             ELSIF (#instMoveSuperimposed.Error = TRUE) THEN
               // Errorhandling
               #statStatus := #ERR_MC_MOVESUPERIMPOSED;
               #statStatusText := STRING#'ERR_MC_MOVESUPERIMPOSED';
               #statErrorAutoCleared := TRUE;
               #statDiagnostics.subfunctionStatus := #statSubfunctionStatus := #instMoveSuperimposed.ErrorID;
               // Set next state
               #statFBState := #AXIS_STOP_ON_ERROR_SELECTION;
               #statSupImpMotionState := #NO_SELECTION;
             ELSE
               ; // command selected
             END_IF;
             #statExeOfSupImpMotionState := 16#0;
             #statExeOfSupImpMotionState.%X0 := #instMoveSuperimposed.Busy;
             #statExeOfSupImpMotionState.%X1 := #instMoveSuperimposed.Done;
             #statExeOfSupImpMotionState.%X2 := #instMoveSuperimposed.CommandAborted;
             #statExeOfSupImpMotionState.%X3 := #instMoveSuperimposed.Error;
             #statExeOfSupImpMotionState.%X4 := #instMoveSuperimposed.Busy;
           END_IF;
         END_REGION

       #PHASING_SELECTED:
         // Additional features (applicative) : Change setpoint on the fly (phaseShift)
         REGION PHASING_SELECTED
           // Firstcycle of command
           IF (#statFirstCycleSupImpMotion = TRUE) THEN
             // Reset MC_PHASING_ABSOLUTE command
             #instPhasingAbsolute(Master := #master,
                                  Slave := #statAxis,
                                  Execute := FALSE);

             // Reset MC_PHASING_RELATIVE command
             #instPhasingRelative(Master := #master,
                                  Slave := #statAxis,
                                  Execute := FALSE);

             #statPhaseShift := #configuration.phasing.phaseShift;
             #statSupImpVelocity := #configuration.phasing.velocity;
             #statSupImpAcceleration := #configuration.phasing.acceleration;
             #statSupImpDeceleration := #configuration.phasing.deceleration;
             #statSupImpJerk := #configuration.phasing.jerk;
             #statSupImpProfileReference := #configuration.phasing.profileReference;
             #statSupImpDistance := #configuration.phasing.phasingDistance;
             #statSupImpStartPosition := #configuration.phasing.startPosition;
             #statSupImpDirection := #configuration.phasing.direction;

             #statPhaseAbsolute := #configuration.phasing.phaseAbsolute;
             #statChangePhaseShiftOnTheFly := #configuration.phasing.phaseShiftChangeOnTheFly;

           ELSIF ((#statChangePhaseShiftOnTheFly = TRUE) AND
             (#configuration.phasing.phaseShift <> #statPhaseShift))
             AND (#statPhaseAbsolute = TRUE)
             AND (#instPhasingAbsolute.CommandAborted = FALSE)
           THEN
             // Reset MC_PHASING_ABSOLUTE command - Phaseshift on the fly is only possible at phasing absolut
             #instPhasingAbsolute(Master := #master,
                                  Slave := #statAxis,
                                  Execute := FALSE);

             #statPhaseShift := #configuration.phasing.phaseShift;

             // V1.0.5 Copy also Dynamics
             #statSupImpVelocity := #configuration.phasing.velocity;
             #statSupImpAcceleration := #configuration.phasing.acceleration;
             #statSupImpDeceleration := #configuration.phasing.deceleration;
             #statSupImpJerk := #configuration.phasing.jerk;
             #statSupImpProfileReference := #configuration.phasing.profileReference;
             #statSupImpDistance := #configuration.phasing.phasingDistance;
             #statSupImpStartPosition := #configuration.phasing.startPosition;
             #statSupImpDirection := #configuration.phasing.direction;

           END_IF;

           // Select phasing absolut or relative 
           IF (#statPhaseAbsolute = TRUE) THEN
             // Absolute phasing
             // Call MC_Command
             #instPhasingAbsolute(Master := #master,
                                  Slave := #statAxis,
                                  Execute := #statSupImpCommand.%X1, // Input: phasing
                                  PhaseShift := #statPhaseShift,
                                  Velocity := #statSupImpVelocity,
                                  Acceleration := #statSupImpAcceleration,
                                  Deceleration := #statSupImpDeceleration,
                                  Jerk := #statSupImpJerk,
                                  ProfileReference := #statSupImpProfileReference,
                                  PhasingDistance := #statSupImpDistance,
                                  StartPosition := #statSupImpStartPosition,
                                  Direction := #statSupImpDirection);

             // Evaluate MC_Command
             IF (#instPhasingAbsolute.Busy = FALSE) AND
               (#instPhasingAbsolute.Error = FALSE) AND
               (#instPhasingAbsolute.Done = FALSE) AND
               (#instPhasingAbsolute.CommandAborted = FALSE)
             THEN
               // Return to NO_SELECTION if command finished
               #statSupImpMotionState := #NO_SELECTION;

             ELSIF (#instPhasingAbsolute.Error = TRUE) THEN
               // Errorhandling
               #statStatus := #ERR_MC_PHASINGABSOLUTE;
               #statStatusText := STRING#'ERR_MC_PHASINGABSOLUTE';
               #statErrorAutoCleared := TRUE;
               #statDiagnostics.subfunctionStatus := #statSubfunctionStatus := #instPhasingAbsolute.ErrorID;
               #statChangePhaseShiftOnTheFly := FALSE;
               // Set next state
               #statFBState := #AXIS_STOP_ON_ERROR_SELECTION;
               #statSupImpMotionState := #NO_SELECTION;
             ELSE
               ; // Command busy
             END_IF;
             #statExeOfSupImpMotionState := 16#0;
             #statExeOfSupImpMotionState.%X0 := #instPhasingAbsolute.Busy;
             #statExeOfSupImpMotionState.%X1 := #instPhasingAbsolute.Done;
             #statExeOfSupImpMotionState.%X2 := #instPhasingAbsolute.CommandAborted;
             #statExeOfSupImpMotionState.%X3 := #instPhasingAbsolute.Error;
             #statExeOfSupImpMotionState.%X4 := #instPhasingAbsolute.StartPhasing;
           ELSE
             // Relative phasing  
             // Call MC_Command
             #instPhasingRelative(Master := #master,
                                  Slave := #statAxis,
                                  Execute := #statSupImpCommand.%X1, // Input: phasing
                                  PhaseShift := #statPhaseShift,
                                  Velocity := #statSupImpVelocity,
                                  Acceleration := #statSupImpAcceleration,
                                  Deceleration := #statSupImpDeceleration,
                                  Jerk := #statSupImpJerk,
                                  ProfileReference := #configuration.phasing.profileReference,
                                  PhasingDistance := #configuration.phasing.phasingDistance,
                                  StartPosition := #configuration.phasing.startPosition,
                                  Direction := #configuration.phasing.direction);

             // Evaluate MC_Command
             IF (#instPhasingRelative.Busy = FALSE) AND
               (#instPhasingRelative.Error = FALSE) AND
               (#instPhasingRelative.Done = FALSE) AND
               (#instPhasingRelative.CommandAborted = FALSE)
             THEN
               // Return to NO_SELECTION if command finished
               #statSupImpMotionState := #NO_SELECTION;

             ELSIF (#instPhasingRelative.Error = TRUE) THEN
               // Errorhandling
               #statStatus := #ERR_MC_PHASINGRELATIVE;
               #statStatusText := STRING#'ERR_MC_PHASINGRELATIVE';
               #statErrorAutoCleared := TRUE;
               #statDiagnostics.subfunctionStatus := #statSubfunctionStatus := #instPhasingRelative.ErrorID;
               #statChangePhaseShiftOnTheFly := FALSE;
               // Set next state
               #statFBState := #AXIS_STOP_ON_ERROR_SELECTION;
               #statSupImpMotionState := #NO_SELECTION;
             ELSE
               ; // Command selected
             END_IF;
             #statExeOfSupImpMotionState := 16#0;
             #statExeOfSupImpMotionState.%X0 := #instPhasingRelative.Busy;
             #statExeOfSupImpMotionState.%X1 := #instPhasingRelative.Done;
             #statExeOfSupImpMotionState.%X2 := #instPhasingRelative.CommandAborted;
             #statExeOfSupImpMotionState.%X3 := #instPhasingRelative.Error;
             #statExeOfSupImpMotionState.%X4 := #instPhasingRelative.StartPhasing;
           END_IF;
         END_REGION

       #OFFSET_SELECTED:
         REGION OFFSET_SELECTED
           // Firstcycle of command
           IF (#statFirstCycleSupImpMotion = TRUE) THEN
             // Reset MC_OFFSET_ABSOLUTE command
             #instOffsetAbsolute(Slave := #statAxis,
                                 Execute := FALSE);

             // Reset MC_OFFSET_RELATIVE command
             #instOffsetRelative(Slave := #statAxis,
                                 Execute := FALSE);

             #statOffsetValue := #configuration.offset.offset;
             #statSupImpProfileReference := #configuration.offset.profileReference;
             #statSupImpDistance := #configuration.offset.offsetDistance;
             #statSupImpStartPosition := #configuration.offset.startPosition;
             #statSupImpDirection := #configuration.offset.direction;

             #statOffsetAbsolute := #configuration.offset.offsetAbsolute;
             #statChangeOffsetOnTheFly := #configuration.offset.offsetChangeOnTheFly;

           ELSIF ((#statChangeOffsetOnTheFly = TRUE) AND
             (#configuration.offset.offset <> #statOffsetValue))
             AND (#statOffsetAbsolute = TRUE)
             AND (#instOffsetAbsolute.CommandAborted = FALSE)
           THEN
             // Reset MC_OFFSET_ABSOLUTE command - Offset on the fly is only possible at phasing absolut
             #instOffsetAbsolute(Slave := #statAxis,
                                 Execute := FALSE);

             #statOffsetValue := #configuration.offset.offset;
           END_IF;

           // Select offset absolut or relative 
           IF (#statOffsetAbsolute = TRUE) THEN
             // Absolute phasing
             // Call MC_Command
             #instOffsetAbsolute(Slave := #statAxis,
                                 Execute := #statSupImpCommand.%X2, // Input: offset
                                 Offset := #statOffsetValue,
                                 ProfileReference := #statSupImpProfileReference,
                                 OffsetDistance := #statSupImpDistance,
                                 StartPosition := #statSupImpStartPosition,
                                 Direction := #statSupImpDirection);

             // Evaluate MC_Command
             IF (#instOffsetAbsolute.Busy = FALSE) AND
               (#instOffsetAbsolute.Error = FALSE) AND
               (#instOffsetAbsolute.Done = FALSE) AND
               (#instOffsetAbsolute.CommandAborted = FALSE)
             THEN
               // Return to NO_SELECTION if command finished
               #statSupImpMotionState := #NO_SELECTION;

             ELSIF (#instOffsetAbsolute.Error = TRUE) THEN
               // Errorhandling
               #statStatus := #ERR_MC_OFFSETABSOLUTE;
               #statStatusText := STRING#'ERR_MC_OFFSETABSOLUTE';
               #statErrorAutoCleared := TRUE;
               #statDiagnostics.subfunctionStatus := #statSubfunctionStatus := #instOffsetAbsolute.ErrorID;
               #statChangeOffsetOnTheFly := FALSE;
               // Set next state
               #statFBState := #AXIS_STOP_ON_ERROR_SELECTION;
               #statSupImpMotionState := #NO_SELECTION;
             ELSE
               ; // Command busy
             END_IF;
             #statExeOfSupImpMotionState := 16#0;
             #statExeOfSupImpMotionState.%X0 := #instOffsetAbsolute.Busy;
             #statExeOfSupImpMotionState.%X1 := #instOffsetAbsolute.Done;
             #statExeOfSupImpMotionState.%X2 := #instOffsetAbsolute.CommandAborted;
             #statExeOfSupImpMotionState.%X3 := #instOffsetAbsolute.Error;
             #statExeOfSupImpMotionState.%X4 := #instOffsetAbsolute.StartOffset;
           ELSE
             // Relative offset  
             // Call MC_Command
             #instOffsetRelative(Slave := #statAxis,
                                 Execute := #statSupImpCommand.%X2, // Input: offset
                                 Offset := #statOffsetValue,
                                 ProfileReference := #configuration.offset.profileReference,
                                 OffsetDistance := #configuration.offset.offsetDistance,
                                 StartPosition := #configuration.offset.startPosition,
                                 Direction := #configuration.offset.direction);

             // Evaluate MC_Command
             IF (#instOffsetRelative.Busy = FALSE) AND
               (#instOffsetRelative.Error = FALSE) AND
               (#instOffsetRelative.Done = FALSE) AND
               (#instOffsetRelative.CommandAborted = FALSE)
             THEN
               // Return to NO_SELECTION if command finished
               #statSupImpMotionState := #NO_SELECTION;

             ELSIF (#instOffsetRelative.Error = TRUE) THEN
               // Errorhandling
               #statStatus := #ERR_MC_OFFSETRELATIVE;
               #statStatusText := STRING#'ERR_MC_OFFSETRELATIVE';
               #statErrorAutoCleared := TRUE;
               #statDiagnostics.subfunctionStatus := #statSubfunctionStatus := #instOffsetRelative.ErrorID;
               #statChangeOffsetOnTheFly := FALSE;
               // Set next state
               #statFBState := #AXIS_STOP_ON_ERROR_SELECTION;
               #statSupImpMotionState := #NO_SELECTION;
             ELSE
               ; // Command selected
             END_IF;
             #statExeOfSupImpMotionState := 16#0;
             #statExeOfSupImpMotionState.%X0 := #instOffsetRelative.Busy;
             #statExeOfSupImpMotionState.%X1 := #instOffsetRelative.Done;
             #statExeOfSupImpMotionState.%X2 := #instOffsetRelative.CommandAborted;
             #statExeOfSupImpMotionState.%X3 := #instOffsetRelative.Error;
             #statExeOfSupImpMotionState.%X4 := #instOffsetRelative.StartOffset;
           END_IF;
         END_REGION
       ELSE
         // Errorhandling
         #statStatus := #ERR_UNDEFINED_SUPERIMPOSED_MOTION_STATE;
         #statStatusText := STRING#'ERR_UNDEFINED_SUPERIMPOSED_MOTION_STATE';
         #statErrorUserCleared := TRUE;
         #statDiagnostics.subfunctionStatus := #statSubfunctionStatus := 0;
         // Set errorstate
         #statFBState := #FB_ERROR;
     END_CASE;
   END_REGION

   //----------------------------------------------------------------------------------------------
   // Execution of torquelimiting functionality
   //----------------------------------------------------------------------------------------------
   REGION EXECUTION_OF_TORQUELIMTING
     // Statemachine for torquelimiting 
     REPEAT
       #tempStateChangeActive := FALSE;
       CASE #statTorqueLimitingState OF
         #NO_TORQUE_LIMITING_ACTIVE:
           ;

         #TORQUE_LIMITING_DISABLE:
           // Torquelimiting disable
           #instTorqueLimiting(Axis := #statAxis,
                               Enable := FALSE);

           // Check state of torque limting
           IF (#instTorqueLimiting.Busy = FALSE)
           THEN
             // set next state
             #statTorqueLimitingState := #NO_TORQUE_LIMITING_ACTIVE;
           ELSE
             ; // Waiting for MC_Torquelimiting is not busy
           END_IF;

         #TORQUE_LIMTING_SELECTED:
           // No extended homing function active
           #instTorqueLimiting(Axis := #statAxis,
                               Enable := #statExtendedCommand.%X1,
                               Limit := #configuration.torqueLimiting.limit,
                               Mode := #configuration.torqueLimiting.mode);

           IF (#instTorqueLimiting.Busy = FALSE) THEN
             // Reset state
             #statTorqueLimitingState := #NO_TORQUE_LIMITING_ACTIVE;
           END_IF;

         #FIXED_STOP_DETECTION_ACTIVE:
           // Extended homing function active
           #instTorqueLimiting(Axis := #statAxis,
                               Enable := TRUE,
                               Limit := #configuration.homing.extendedModeTorqueLimit, // V01.00.03 Always use configured value
                               Mode := #MODE_FIXED_STOP_DETECTION);

           IF ((#statHomingSubState = #HOMING_IDLE) AND (#statBasicMotionState = #ACTIVE_HOMING_SELECTED))
           THEN
             // Fixed stop process has finished - Axis is still in clamping
             #statTorqueLimitingState := #FIXED_STOP_DETECTION_FINISHED;
             #tempStateChangeActive := TRUE;

           ELSIF (#statBasicMotionState <> #ACTIVE_HOMING_SELECTED)
           THEN
             // Error occurred - change state depending on inClamping
             IF (#instTorqueLimiting.InClamping = TRUE)
             THEN
               // Axis is in clamping
               #statTorqueLimitingState := #FIXED_STOP_DETECTION_ERROR_IN_CLAMPING;
               #tempStateChangeActive := TRUE;
             ELSE
               // Axis is in not clamping
               #statTorqueLimitingState := #FIXED_STOP_DETECTION_ERROR_NOT_IN_CLAMPING;
               #tempStateChangeActive := TRUE;
             END_IF;
           ELSE
             ; // Fixed stop detection is running
           END_IF;

         #FIXED_STOP_DETECTION_FINISHED:
           // Homing on fixed stop process has finished
           #instTorqueLimiting(Axis := #statAxis,
                               Enable := TRUE,
                               Limit := #configuration.homing.extendedModeTorqueLimit, // V01.00.03 Always use configured value
                               Mode := #MODE_FIXED_STOP_DETECTION);

           IF (#instTorqueLimiting.InClamping = FALSE)
           THEN
             // InClamping = FALSE
             IF (#statExtendedCommand.%X1 = TRUE) // Torquelimiting
             THEN
               #statTorqueLimitingState := #TORQUE_LIMTING_SELECTED;
             ELSE
               #statTorqueLimitingState := #TORQUE_LIMITING_DISABLE;
             END_IF;
             #tempStateChangeActive := TRUE;
           ELSE
             // InClamping = TRUE
             IF (#statExtendedCommand.%X1 = TRUE) // Torquelimiting
               AND (#configuration.torqueLimiting.mode = #MODE_FIXED_STOP_DETECTION)
             THEN
               // Change State
               #statTorqueLimitingState := #TORQUE_LIMTING_SELECTED;
               #tempStateChangeActive := TRUE;
             ELSE
               ; // Wait for inClamping = FALSE
             END_IF;
           END_IF;

         #FIXED_STOP_DETECTION_ERROR_IN_CLAMPING:
           // Errorstate, torquelimiting is still active and axis not in clamping
           #instTorqueLimiting(Axis := #statAxis,
                               Enable := TRUE,
                               Limit := #configuration.homing.extendedModeTorqueLimit, // V01.00.03 Always use configured value
                               Mode := #MODE_FIXED_STOP_DETECTION);

           IF (#instTorqueLimiting.InClamping = FALSE)
           THEN
             // InClamping = FALSE -> reset torque limiting state
             #statTorqueLimitingState := #TORQUE_LIMITING_DISABLE;
             // Torquelimiting disable
             #tempStateChangeActive := TRUE;
           END_IF;

         #FIXED_STOP_DETECTION_ERROR_NOT_IN_CLAMPING:
           // Errorstate, torquelimiting is still active and axis in clamping
           #instTorqueLimiting(Axis := #statAxis,
                               Enable := TRUE,
                               Limit := #configuration.homing.extendedModeTorqueLimit, // V01.00.03 Always use configured value
                               Mode := #MODE_FIXED_STOP_DETECTION);

           IF (#instTorqueLimiting.InClamping = TRUE)
           THEN
             // InClamping = TRUE -> change state
             #statTorqueLimitingState := #FIXED_STOP_DETECTION_ERROR_IN_CLAMPING;
             #tempStateChangeActive := TRUE;

           ELSIF (#statBasicMotionState <> #NO_SELECTION)
             OR (#statSupImpMotionState <> #NO_SELECTION)
             OR (#statPassiveHomingState <> #NO_HOMING_ACTIVE)
           THEN
             // New valid command is set -> reset error state
             #statTorqueLimitingState := #TORQUE_LIMITING_DISABLE;
             #tempStateChangeActive := TRUE;
           ELSE
             ; // Waiting for new command or axis is getting in clamping
           END_IF;
         ELSE
           // Errorhandling
           #statStatus := #ERR_UNDEFINED_TORQUE_LIMITING_STATE;
           #statStatusText := STRING#'ERR_UNDEFINED_TORQUE_LIMITING_STATE';
           #statErrorUserCleared := TRUE;
           #statDiagnostics.basicMotionState := #statBasicMotionState;
           #statDiagnostics.superimposedMotionState := #statSupImpMotionState;
           #statDiagnostics.subfunctionStatus := #statSubfunctionStatus := 0;
           // Set errorstate
           #statFBState := #FB_ERROR;
       END_CASE;
     UNTIL (#tempStateChangeActive = FALSE)
     END_REPEAT;
     // Evaluate MC_Command
     IF (#instTorqueLimiting.Error = TRUE) AND ((#statTorqueLimitingErrorOld = FALSE) OR (#statStatus = #STATUS_SUBSEQUENT_CALL)) THEN
       // Errorhandling
       #statStatus := #ERR_MC_TORQUELIMITING;
       #statStatusText := STRING#'ERR_MC_TORQUELIMITING';
       #statErrorAutoCleared := TRUE;
       #statDiagnostics.basicMotionState := #statBasicMotionState;
       #statDiagnostics.superimposedMotionState := #statSupImpMotionState;
       #statDiagnostics.subfunctionStatus := #statSubfunctionStatus := #instTorqueLimiting.ErrorId;

       #statFBState := #AXIS_STOP_ON_ERROR_SELECTION;

     ELSIF (#instTorqueLimiting.Error = FALSE) AND ((#statTorqueLimitingErrorOld = TRUE) AND (#statStatus = #ERR_MC_TORQUELIMITING)) THEN
       #statStatus := #STATUS_SUBSEQUENT_CALL;
       #statStatusText := STRING#'STATUS_SUBSEQUENT_CALL';
       #statErrorAutoCleared := FALSE;
     ELSE
       ;
     END_IF;

     #statTorqueLimitingErrorOld := #instTorqueLimiting.Error;
   END_REGION

   //----------------------------------------------------------------------------------------------
   // Selection of StopOnError / implementation of fastStop
   //----------------------------------------------------------------------------------------------
   REGION STOP_ON_ERROR
     // Check for stopping if error occurred during execution of motion commands
     IF (#statFBState = #AXIS_STOP_ON_ERROR_SELECTION)
     THEN
       #statBasicMotionState := #NO_SELECTION;
       #statSupImpMotionState := #NO_SELECTION;
       #statPassiveHomingState := #NO_HOMING_ACTIVE;

       IF (#configuration.generalSettings.stopOnError = TRUE)
       THEN
         // Read Statusword
         #tempStatusWord := "LAxisCtrl_UnpubAxisStatusWord"(#statAxis);

         // Evaluate error
         IF #tempStatusWord.%X0 THEN
           // Axis enabled
           IF (#tempStatusWord.%X1 = TRUE) THEN
             // TO Alarm present
             #statFBState := #AXIS_MOTION;
           ELSE
             // No TO alarm present, set fastStop
             //#statBasicMotionState := #FAST_STOP_SELECTED; // V1.1.0
             #statStopWithoutSignalization := TRUE; // V1.1.0
             #statFirstCycleBasicMotion := TRUE;
             #statFBState := #AXIS_STOP_ON_ERROR_EXECUTION;
           END_IF;
         ELSE
           // Axis disabled
           #statFBState := #AXIS_MOTION;
         END_IF;
       ELSE
         // Dont StopOnError
         #statFBState := #AXIS_MOTION;
       END_IF;
     END_IF;

     // Implementation of fastStop
     IF #statStopWithoutSignalization
       OR
       (
       TRUE
       AND (#statBasicMotionState = #FAST_STOP_SELECTED)
       AND (#statMainSelectionState = #CALL_BASIC_MOTION)
       )
     THEN
       // Additional feature: Load emergency stop dynamics (TO) if no valid dynamics are configured for fastStop
       REGION FASTSTOP SELECTED
         // Firstcycle of command
         IF (#statFirstCycleBasicMotion = TRUE) THEN
           // Reset HALT command
           #instHalt(Axis := #statAxis,
                     Execute := FALSE);
           #statFirstCycleDone := TRUE;
           // Check dynamics for fastStop
           // Load TO emergency Stop dynamics if value <=0 for deceleration is configured
           IF (#configuration.fastStop.deceleration <= 0.0) // V1.0.2 Read TO emergencyStop deceleration only if fastStop.deceleration <= 0
           THEN
             // Invalid fastStop dynamics configured - read emergency stop dynamics from TO
             #statBasicDeceleration := "LAxisCtrl_UnpubAxisEmergencyDec"(#statAxis);
           ELSE
             // Valid fastStop dynamics configured
             #statBasicDeceleration := #configuration.fastStop.deceleration;
           END_IF;
           #statBasicJerk := #configuration.fastStop.jerk; // V1.0.2 Use always configuration for jerk value
           #statBasicAbortAcceleration := #configuration.fastStop.abortAcceleration; // V1.0.2 Use always configuration
         END_IF;

         // Call of MC_Command
         #instHalt(Axis := #statAxis,
                   Execute := (#statBasicCommand.%X0 OR #statFirstCycleBasicMotion),
                   Deceleration := #statBasicDeceleration,
                   AbortAcceleration := #statBasicAbortAcceleration,
                   Jerk := #statBasicJerk);

         // Evaluate MC_Command
         IF (#instHalt.Busy = FALSE) AND
           (#instHalt.Error = FALSE) AND
           (#instHalt.Done = FALSE) AND
           (#instHalt.CommandAborted = FALSE)
         THEN
           // Return to NO_SELECTION if command finished
           #statFBState := #AXIS_MOTION;
           #statBasicMotionState := #NO_SELECTION;
           #statStopWithoutSignalization := FALSE; // V1.1.0

         ELSIF (#instHalt.Done = TRUE)
         THEN
           IF (#statFirstCycleDone = TRUE)
           THEN
             // Command is reset
             IF (#instTorqueLimiting.Error = FALSE) // V1.00.03 Dont reset error is pending
             THEN
               // Reset status not if torquelimiting error is pending
               IF #statStopWithoutSignalization THEN
                 ;
               ELSE
                 #statStatus := #STATUS_SUBSEQUENT_CALL;
                 #statStatusText := STRING#'STATUS_SUBSEQUENT_CALL';
                 #statErrorAutoCleared := FALSE;
               END_IF;
             END_IF;

             #statFirstCycleDone := FALSE;
           END_IF;
         ELSE
           ; // Command selected
         END_IF;

         // Write MC_Command outputs to internal variable
         #statExeOfBasicMotion := 0;
         #statExeOfBasicMotion.%X0 := #instHalt.Busy;
         #statExeOfBasicMotion.%X1 := #instHalt.Done;
         #statExeOfBasicMotion.%X2 := #instHalt.CommandAborted;
         #statExeOfBasicMotion.%X3 := #instHalt.Error;
       END_REGION
     END_IF;
   END_REGION
   //----------------------------------------------------------------------------------------------
   // Store values and reset variables
   //----------------------------------------------------------------------------------------------
   REGION STORE_AND_RESET
     // Reset variables to determine first cycle of a new command
     IF (#statFirstCycleReset = TRUE) THEN
       #statFirstCycleReset := FALSE;
     END_IF;
     IF (#statFirstCycleHoming = TRUE) THEN
       #statFirstCycleHoming := FALSE;
     END_IF;
     #statHomingOld := #tempHoming;

     #statFirstCycleBasicMotion := FALSE;
     #statBasicCommandOld := #statBasicCommand;

     IF (#statFirstCycleSupImpMotion = TRUE) THEN
       #statFirstCycleSupImpMotion := FALSE;
     END_IF;
     #statSupImpCommandOld := #statSupImpCommand;

     // Store last values for edge detection
     #statEnableOld := #tempEnable;
     #statEnableAxisOld := #tempEnableAxis;
     #statExtendedCommandOld := #statExtendedCommand;
     #statPowerErrorOld := #instPower.Error;
   END_REGION

   //----------------------------------------------------------------------------------------------
   // Writing outputs
   //----------------------------------------------------------------------------------------------
   REGION WRITING_OF_OUTPUTS
     // Writing status outputs
     #resetActive := (#statResetState = #CMD_BUSY);

     IF (#statErrorUserCleared = TRUE) THEN
       ; // Reset variables at ErrorUserCleared
       #statBasicMotionState := #NO_SELECTION;
       #statExeOfBasicMotion := #NO_SELECTION;
       #statSupImpMotionState := #NO_SELECTION;
       #statExeOfSupImpMotionState := #NO_SELECTION;
       #statExeOfHoming := #NO_SELECTION;
     END_IF;
     IF (#instPower.Status = TRUE)
     THEN
       // Axis enabled
       #axisEnabled := TRUE;

     ELSIF (#instPower.Error = TRUE) AND (#instPower.Status = FALSE)
     THEN
       // Reset status if error occurred
       #axisEnabled := FALSE;

     ELSIF (#instPower.Busy = FALSE)
     THEN
       // Reset if MC_Power is not busy
       #axisEnabled := FALSE;
     ELSE
       ;
     END_IF;

     REGION WRITING_BASICMOTION_OUTPUTS
       // Writing Busy, Done and Aborted outputs for basic motion commands
       IF (#statBasicMotionState > #NO_SELECTION) AND (#statBasicMotionState <> #ACTIVE_HOMING_SELECTED)
       THEN
         #commandBusy := #statExeOfBasicMotion.%X0;
         #commandDone := #statExeOfBasicMotion.%X1;
         #commandAborted := #statExeOfBasicMotion.%X2;
         #inVelocity := #statExeOfBasicMotion.%X4;
         #inSync := #statExeOfBasicMotion.%X7;
         #startSync := #statExeOfBasicMotion.%X6;
         #endOfProfile := #statExeOfBasicMotion.%X8;
       ELSE
         #commandBusy := FALSE;
         #commandDone := FALSE;
         #commandAborted := FALSE;
         #inVelocity := FALSE;
         #inSync := FALSE;
         #startSync := FALSE;
         #endOfProfile := FALSE;
       END_IF;

       // Writing outputs up to LAxisCtrl_SpeedAxis
       IF (#statTorqueLimitingState = #TORQUE_LIMTING_SELECTED)
         // OR (#statTorqueLimitingState = #AUTOMATIC_MODE_CHANGE) V1.0.3 TorqueLimtinig = TRUE, only when respective value used 
       THEN
         #torqueLimitingSelected := TRUE;
       ELSE
         #torqueLimitingSelected := FALSE;
       END_IF;

       #inLimitation := #instTorqueLimiting.InLimitation;
       #fastStopSelected := #statBasicMotionState.%X0;
       #stopSelected := #statBasicMotionState.%X1;
       #jogSelected := #statBasicMotionState.%X2 OR #statBasicMotionState.%X3;
       #moveVelocitySelected := #statBasicMotionState.%X4;
       // Writing outputs up to LAxisCtrl_PosAxis
       #inClamping := #instTorqueLimiting.InClamping;
       #posRelativeSelected := #statBasicMotionState.%X5;
       #posAbsoluteSelected := #statBasicMotionState.%X6;
       // Writing outputs up to LAxisCtrl_SyncAxisRelGearing
       #gearInRelativeSelected := #statBasicMotionState.%X7;
       // Writing outputs up to LAxisCtrl_SyncAxisCamming
       #gearInAbsoluteSelected := #statBasicMotionState.%X8;
       #camInSelected := #statBasicMotionState.%X9;
       #gearOutCamOutSelected := #statBasicMotionState.%X11;
       #inSimulation := #instSyncMotionSimulation.InSimulation;
     END_REGION
     REGION WRITING_HOMING_OUTPUTS
       // Writing Busy, Done and Aborted outputs for homing
       IF (#statPassiveHomingState = #STANDARD_HOMING)
       THEN
         #homingSelected := TRUE;
         #homingCommandBusy := #statExeOfHoming.%X0;
         #homingCommandDone := #statExeOfHoming.%X1;
         #homingCommandAborted := #statExeOfHoming.%X2;
       ELSE
         IF (#statBasicMotionState = #ACTIVE_HOMING_SELECTED)
         THEN
           #homingSelected := TRUE;
           #homingCommandBusy := #statExeOfBasicMotion.%X0;
           #homingCommandDone := #statExeOfBasicMotion.%X1;
           #homingCommandAborted := #statExeOfBasicMotion.%X2;
         ELSE
           #homingSelected := FALSE;
           #homingCommandBusy := FALSE;
           #homingCommandDone := FALSE;
           #homingCommandAborted := FALSE;
         END_IF;
       END_IF;
     END_REGION
     REGION WRITING_SUPERIMPOSED_OUTPUTS
       // Writing outputs for superimposed motion commands
       IF (#statSupImpMotionState <> #NO_SELECTION)
       THEN
         #superimposedBusy := #statExeOfSupImpMotionState.%X0;
         #superimposedDone := #statExeOfSupImpMotionState.%X1;
         #superimposedAborted := #statExeOfSupImpMotionState.%X2;
         #superimposedStart := #statExeOfSupImpMotionState.%X4;
       ELSE
         #superimposedBusy := FALSE;
         #superimposedDone := FALSE;
         #superimposedAborted := FALSE;
         #superimposedStart := FALSE;
       END_IF;
       #posSuperimposedSelected := #statSupImpMotionState.%X0;
       #phasingSelected := #statSupImpMotionState.%X1;
       #offsetSelected := #statSupImpMotionState.%X2;
     END_REGION
   END_REGION

   //----------------------------------------------------------------------------------------------
   // Error handling 
   //----------------------------------------------------------------------------------------------
   REGION ERROR_HANDLING
     IF #statErrorUserCleared THEN
       #valid := FALSE;
       #busy := TRUE;
       #error := TRUE;
       #subfunctionStatus := #statSubfunctionStatus; // V1.1.0
       #statDiagnostics.status := #statStatus;

     ELSIF #statErrorAutoCleared THEN
       #valid := FALSE;
       #busy := TRUE;
       #error := TRUE;
       #subfunctionStatus := #statSubfunctionStatus; // V1.1.0
       #statDiagnostics.status := #statStatus;

     ELSE
       // Process normal output values
       #valid := TRUE;
       #error := FALSE;
       #subfunctionStatus := #statSubfunctionStatus := 16#0; // V1.1.0
     END_IF;

     #status := #statStatus;

     IF (#statStatus <> #statStatusOld) THEN
       #statusText := #statStatusText;   // V1.2.0
       #diagnostics := #statDiagnostics; // V1.1.0
     END_IF;

     // Edge detection
     #statStatusOld := #statStatus;
   END_REGION
END_FUNCTION_BLOCK